// TwinCAT 3 PLC project beckhoffTutorial01
// ProgramVersion: 3.1.4024.0
// libraries:
//   Tc2_Math, * (Beckhoff Automation GmbH)
//   Tc2_Standard, * (Beckhoff Automation GmbH)
//   Tc2_System, * (Beckhoff Automation GmbH)
//   Tc3_Analytics, * (Beckhoff Automation GmbH)
//   Tc3_Module, * (Beckhoff Automation GmbH)
//   VisuSymbols,3.5.10.0,System
// project tree:
//   / GlobalTextList.TcGTLO, PlcTask.TcTTO, Visualization Manager.TcVMO (not stored)
//   GVLs/ GVL.TcGVL
//   POUs/ f_mmToInch.TcPOU, InstrumentReading_420mA.TcPOU, MAIN.TcPOU
//   VISUs/ PositionTrans.TcVIS
// real-time tasks:
//   TASK PlcTask: cycle T#10ms, priority 20, ADS port 350
// I/O:
//   DEVICE Device 1 (EtherCAT), AmsNetId 5.141.19.14.2.1
//     Term 1 (EK1200) [EK1200-5000 EtherCAT Power supply (2A E-Bus)]
//       Term 2 (EL1809) [EL1809 16Ch. Dig. Input 24V, 3ms]
//       Term 3 (EL3114) [EL3114 4Ch. Ana. Input 0-20mA Diff.]
//       Term 4 (EL3104) [EL3104 4Ch. Ana. Input +/-10V Diff.]
//       Term 5 (EL9011) [EL9011 End Terminal]
// variable links:
//   beckhoffTutorial01/beckhoffTutorial01 Instance <-> Device 1 (EtherCAT)/Term 1 (EK1200)/Term 3 (EL3114)
//     PlcTask Inputs/GVL.nCurrent_Input1 <-> AI Standard Channel 1/Value

CONFIGURATION beckhoffTutorial01
    RESOURCE PLC ON TwinCAT3
        TASK PlcTask(INTERVAL := T#10ms, PRIORITY := 20);
        PROGRAM MAIN WITH PlcTask : MAIN;
    END_RESOURCE
END_CONFIGURATION

// ---- GVLs/GVL.TcGVL
{attribute 'qualified_only'}
VAR_GLOBAL
(* Digital Input variables for EL1809 *)
bDigital_Input1 AT %I* : BOOL;
bDigital_Input2 AT %I* : BOOL;
bDigital_Input3 AT %I* : BOOL;
bDigital_Input4 AT %I* : BOOL;
bDigital_Input5 AT %I* : BOOL;
bDigital_Input6 AT %I* : BOOL;
bDigital_Input7 AT %I* : BOOL;
bDigital_Input8 AT %I* : BOOL;
bDigital_Input9 AT %I* : BOOL;
bDigital_Input10 AT %I* : BOOL;
bDigital_Input11 AT %I* : BOOL;
bDigital_Input12 AT %I* : BOOL;
bDigital_Input13 AT %I* : BOOL;
bDigital_Input14 AT %I* : BOOL;
bDigital_Input15 AT %I* : BOOL;
bDigital_Input16 AT %I* : BOOL;

(*4-20 mA Analog inputs for EL3114*)
nCurrent_Input1 AT %I* : INT;
nCurrent_Input2 AT %I* : INT;
nCurrent_Input3 AT %I* : INT;
nCurrent_Input4 AT %I* : INT;

//Converted from DAQ resolution to engineering unit (mA)
rCurrent_Input1_EU AT %I* : REAL;
rCurrent_Input2_EU AT %I* : REAL;
rCurrent_Input3_EU AT %I* : REAL;
rCurrent_Input4_EU AT %I* : REAL;

(*0-10V Analog Input for EL3104*)
nVoltage_Input1 AT %I* : INT;
nVoltage_Input2 AT %I* : INT;
nVoltage_Input3 AT %I* : INT;
nVoltage_Input4 AT %I* : INT;

//Converted from DAQ resolution to engineering unit (V)
rVoltage_Input1_EU AT %I* : REAL;
rVoltage_Input2_EU AT %I* : REAL;
rVoltage_Input3_EU AT %I* : REAL;
rVoltage_Input4_EU AT %I* : REAL;
END_VAR

// ---- POUs/MAIN.TcPOU
PROGRAM MAIN
VAR
	rPosSenDis_mm : REAL;
	rPosSenDis_inch : REAL;
END_VAR

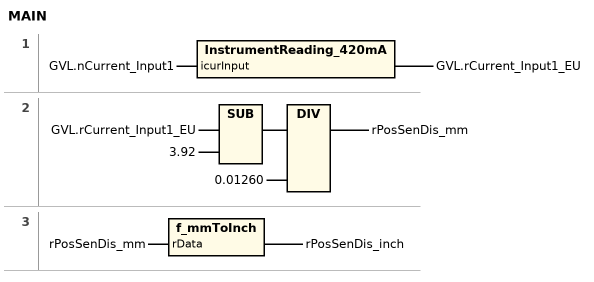
// NETWORK 1
GVL.rCurrent_Input1_EU := InstrumentReading_420mA(icurInput := GVL.nCurrent_Input1);

// NETWORK 2
rPosSenDis_mm := (GVL.rCurrent_Input1_EU - 3.92) / 0.01260;

// NETWORK 3
rPosSenDis_inch := f_mmToInch(rData := rPosSenDis_mm);

END_PROGRAM

// ---- POUs/InstrumentReading_420mA.TcPOU
FUNCTION InstrumentReading_420mA : REAL
(*
* Takes the DAQ's curInput (unitless) and coverts to EU (mA)
* Built for use with EL3114 15 bit resolution
* Change internal variable 
* @param icurInput (INT): Raw data from ADC
* Output rcurOutput (REAL): EU real output
*)
VAR_INPUT
	icurInput : INT;
END_VAR
VAR
	rconvFactor : REAL := 16.0/(26300.0); //Will also convert int to real
END_VAR

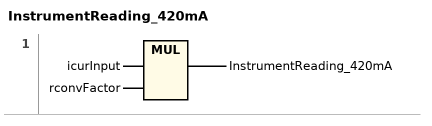
// NETWORK 1
InstrumentReading_420mA := icurInput * rconvFactor;

END_FUNCTION

// ---- POUs/f_mmToInch.TcPOU
FUNCTION f_mmToInch : REAL
VAR_INPUT
	rData : REAL;
END_VAR
VAR
END_VAR

f_mmToInch := rData * 0.0393701;

END_FUNCTION

// ---- GlobalTextList.TcGTLO
TEXTLIST GlobalTextList
  862 = '%'
  636 = '%.2f'
  558 = '%.3f'
  467 = '%.3f inches'
  663 = '%.3f mA'
  721 = '%.3f mm'
  628 = '%lf'
  222 = 'Current value: %5.2f'
  12 = 'Current value: %r'
  142 = 'Position Transducer Reading (mA)'
  704 = 'Position Transducer Reading (mA): %5.2f'
  908 = 'Position Transducer Reading (mA): %lf'
END_TEXTLIST

// ---- VISUs/PositionTrans.TcVIS
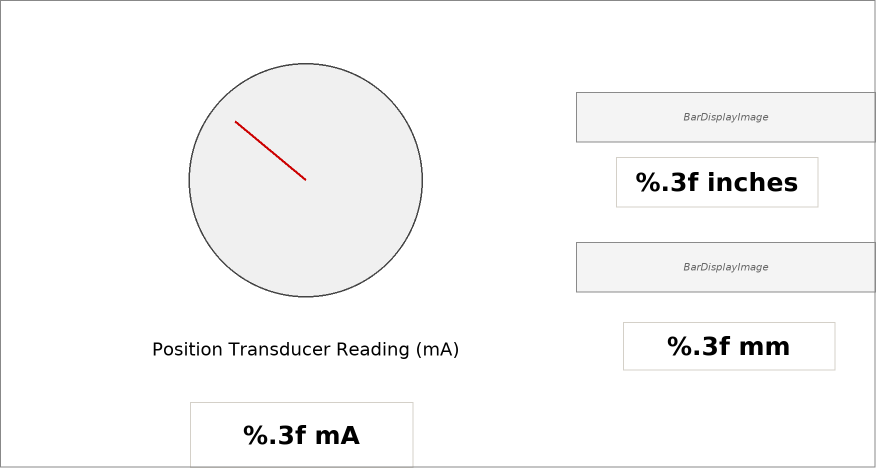
VISUALIZATION PositionTrans  // 876x468
    Meter360 (187,63 237x234), value: GVL.rCurrent_Input1_EU, style: Meter-Meter360-Gray, scale format: %.1f, scale 0..20
    Textfield (128,315 356x69), "Position Transducer Reading (mA)"
    Textfield (190,402 223x66), "%.3f mA", text variable: GVL.rCurrent_Input1_EU
    BarDisplayImage (576,92 300x50), style: BarDisplayImage-Gray, scale format: %.1f, scale 0..100
    BarDisplayImage (576,242 300x50), style: BarDisplayImage-Gray, scale format: %.1f, scale 0..100
    Textfield (616,157 202x50), "%.3f inches", text variable: MAIN.rPosSenDis_inch
    Textfield (623,322 212x48), "%.3f mm", text variable: MAIN.rPosSenDis_mm
END_VISUALIZATION
